TYPE ST_peakshavebox_params :
STRUCT
	ExtBreakerControl	: BOOL := FALSE; 
END_STRUCT
END_TYPE

(* stored: Version 1.1.0.1, ProductVersion 3.1.4026.18
   DUT ST_peakshavebox_params: Id {905fe61c-a96c-43f5-9976-24ad1ecff638} *)
